ABB RobotStudio station: CellaRobotizzata.rspag

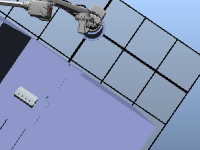
--- station ---
Station Solution8 (saved by RobotStudio 7.0.8504.151)
Controller IRB_4600_20kg_2.50m, task T_ROB1: task frame (RAPID world) sits at (0, 0, 900) mm in the station
Controller IRB_4600_20kg_2.50m
  mechanical unit ROB_1: IRB4600_20_250_C_01, 6 joints, base frame (0, 0, 0) mm
Layout (positions relative to the parent item):
  - IRB4600_20_250_C_01 [mechanism, from Robots\IRB4600_20_250_C_G_01.rslib] at (0, 0, 900) mm; joint values [-1.0848, 0.7462, -0.6696, 1.0226, 1.1134, -1.3841] (rad or m)
  - CentroDiLavoro [part] at (1081.98, 2085.34, 0) mm, rotated rx 90 ry 0 rz -90 deg
  - PalletLavoro [part] at (1981.98, -173.66, 1318.5) mm
  - PalletLavoro_2 [part] at (1081.98, -173.66, 1318.5) mm
  - Basamento_robot_2 [part] at (0, 0, 900) mm
  - testata_motore [part] at (2148.67, -143.24, 1898.49) mm, rotated rx 90 ry 0 rz 0 deg

--- Backups/IRB_4600_20kg_2.50m/RAPID/TASK1/PROGMOD/Module1.mod ---
MODULE Module1
    !***********************************************************
    !
    ! Modulo:  Module1
    !
    ! Descrizione:
    !   <Inserire descrizione qui>
    !
    ! Autore: campr
    !
    ! Versione: 1.0
    !
    !***********************************************************


    !***********************************************************
    !
    ! Procedura main
    !
    !   Questo è il punto di ingresso del programma
    !
    !***********************************************************
    PROC main()
        !Aggiungere il codice in questo punto
    ENDPROC
ENDMODULE
